FUNCTION_BLOCK Path EXTENDS Spline
VAR_INPUT
	waypointListRaw: 	ARRAY [0..100] OF RobotPoseSimple;
	radius: 			LREAL;
	thetaDZ: 				LREAL := 0.1;
END_VAR
VAR
	waypointList: 		ARRAY [0..100] 	OF 	RobotPoseSimple;		
	subsplines: 		ARRAY [0..99] 	OF  POINTER TO Spline;
	transitions: 		ARRAY [0..99] 	OF LREAL;
	nmbOfSubsplines, nmbOfPreprocessedWaypoints:	INT;
END_VAR

preprocessWaypointlist();

nmbOfSubsplines := 2*nmbOfPreprocessedWaypoints-3;

generateSubsplines();
lengthVar := calculateLength();
calculateTransitions();

startPoint := subsplines[0]^.startPointVal;
endPoint   := subsplines[nmbOfSubsplines-1]^.endPointVal;

startPoint.theta := waypointList[0].theta;
endPoint.theta	 := waypointList[nmbOfPreprocessedWaypoints-1].theta;

(* 
Implementation of abstract Spline method.
For internal inital length calculation, should be called in the constructor => protected
*)
METHOD PROTECTED  calculateLength : LREAL
VAR_INPUT
END_VAR
VAR
	i: INT;
END_VAR
calculateLength := 0;
FOR i := 0 TO nmbOfSubsplines-1 DO
	calculateLength := calculateLength + subsplines[i]^.length;
END_FOR
END_METHOD

METHOD PRIVATE calculateTransitions
VAR_INPUT
END_VAR
VAR
	i : INT;
END_VAR
transitions[0] := 0;
FOR i := 0 TO nmbOfSubsplines-2 DO
	transitions[i+1] := transitions[i] + subsplines[i]^.length;
END_FOR
END_METHOD

(* 
Implementation of abstract Spline method.
Calculates the derivate of the spline at an arbitrary arcLength. Should be implmented for order one and two. Invalid 
orders should write a -1 in every component of the return value.
*)
METHOD  PUBLIC diff : RobotPoseSimple
VAR_INPUT
	arcLength: LREAL; //arcLength at which the corresponding derivative should be calculated
	order: INT := 1;  //optional: order of the derivate, should be implemented for 1 and 2, default: 1
END_VAR
VAR
	subspline: 				POINTER TO Spline;
	arcOffset, deltaTheta: 	LREAL;
	dPos: RobotPoseSimple;
END_VAR
getSubsplineToPoint(arcLength := arcLength,
					subspline => subspline,
					arcOffset => arcOffset);
deltaTheta:= endPoint.theta - startPoint.theta; 		
diff 		:= subspline^.diff(arcLength := arcOffset, order:= order);	
diff.theta 	:= dTheta(arcLength := arcLength, order := order);
END_METHOD

METHOD PRIVATE dTheta : LREAL
VAR_INPUT
	arcLength: LREAL;
	order: INT;
END_VAR
VAR
	deltaTheta: LREAL;
END_VAR
deltaTheta := endPoint.theta - startPoint.theta;
IF arcLength < thetaDZ  OR arcLength > lengthVar - thetaDZ THEN
	dTheta := 0;
ELSIF order = 1 THEN
	dTheta := deltaTheta/2*(pi/(lengthVar-2*thetaDZ))*SIN(pi/(lengthVar-2*thetaDZ)*(arcLength-thetaDZ));
ELSIF order = 2 THEN
	dTheta := deltaTheta/2*EXPT(pi/(lengthVar-2*thetaDZ),2)*COS(pi/(lengthVar-2*thetaDZ)*(arcLength-thetaDZ));
END_IF
END_METHOD

METHOD generateSubsplines : BOOL
VAR_INPUT
END_VAR
VAR
	linearSplines:		ARRAY [0..50] OF LinearSpline;
	bezierCurves:		ARRAY [0..49] OF BezierCurve;
		
	//xTmpLinear,yTmpLinear:    		ARRAY [0..1] OF LREAL;
	wplTmpLinear:					ARRAY [0..1] OF RobotPoseSimple;
	linearSpline: LinearSpline;
	
	//xTmpBezier,yTmpBezier:    		ARRAY [0..2] OF LREAL;
	wplTmpBezier:					ARRAY [0..2] OF RobotPoseSimple;
	bezierCurve: BezierCurve;
	
	i,j,k: INT := 0;
END_VAR
IF nmbOfSubsplines <> 1 THEN 
	FOR i := 1 TO nmbOfSubsplines BY 2 DO
	k := 0;
	//extract relevant points for bezier curve creation
	FOR j := (i-1)/2 TO (i-1)/2+2 BY 1 DO
		wplTmpBezier[k] := waypointList[j];
		k := k + 1;
	END_FOR  
	bezierCurves[(i-1)/2](waypoints:=wplTmpBezier, radius:=radius);
	subsplines[i]:= ADR(bezierCurves[(i-1)/2]);
	END_FOR
	
	//first Segment is always linear
	wplTmpLinear[0] := waypointList[0];
	wplTmpLinear[1] := subsplines[1]^.startPointVal;
	linearSplines[0](wayPoints := wplTmpLinear);
	subsplines[0] := ADR(linearSplines[0]);
	
	
	//last Segment is always linear
	wplTmpLinear[0] := subsplines[nmbOfSubsplines-2]^.endPointVal;
	wplTmpLinear[1] := waypointList[nmbOfPreprocessedWaypoints-1];
	linearSplines[(nmbOfSubsplines+1)/2](wayPoints := wplTmpLinear);
	subsplines[nmbOfSubsplines-1] := ADR(linearSplines[(nmbOfSubsplines+1)/2]);
	
	
	//generate the linear segments in between
	FOR i := 2 TO nmbOfSubsplines-2 BY 2 DO
	wplTmpLinear[0] := subsplines[i-1]^.endPointVal;
	wplTmpLinear[1] := subsplines[i+1]^.startPointVal;
	linearSplines[i/2](wayPoints := wplTmpLinear);
	subsplines[i] := ADR(linearSplines[i/2]);
	END_FOR
ELSE  //nmbOfSubsplines = 1  => only one linear Segment
	
	wplTmpLinear[0] := waypointList[0];
	wplTmpLinear[1] := waypointList[1];;
	linearSplines[0](wayPoints := wplTmpLinear);
	subsplines[0] := ADR(linearSplines[0]);
END_IF
END_METHOD

(*
Implementation of abstract Spline method.
Gets the configuration of the Spline at any given arcLength. 
*)
METHOD PUBLIC  getPoint : RobotPoseSimple
VAR_INPUT
	arcLength: LREAL; //arcLength at which the Splines configuration shall be calculated.
END_VAR
VAR
	subspline: POINTER TO Spline;
	arcOffset: LREAL;
	deltaTheta: LREAL;
END_VAR
getSubsplineToPoint(arcLength := arcLength,
					subspline => subspline,
					arcOffset => arcOffset);
getPoint := subspline^.getPoint(arcLength:= arcOffset);

deltaTheta 		:= endPoint.theta - startPoint.theta;
getPoint.theta	:= theta(arcLength := arcLength);
END_METHOD

METHOD PRIVATE getSubsplineToPoint : POINTER TO Spline
VAR_INPUT
	arcLength: LREAL;
END_VAR

VAR_OUTPUT
	subspline: 	POINTER TO Spline;
	arcOffset: 	LREAL;
	i: 			INT := 0;
END_VAR
arcOffset := arcLength;
IF arcLength >= length THEN
	arcOffset := arcLength - transitions[nmbOfSubsplines-1];
	subspline := subsplines[nmbOfSubsplines-1];
	RETURN;
END_IF

FOR i := 0 TO nmbOfSubsplines-1 DO
	IF arcOffset-subsplines[i]^.length < 0 THEN
		subspline := subsplines[i];
		EXIT;
	ELSE
		arcOffset := arcOffset -subsplines[i]^.length;
	END_IF
END_FOR
END_METHOD

METHOD getSwitchingPointIntervals : ARRAY [0..98] OF LREAL
VAR_INPUT
END_VAR
VAR
	i: INT := 0;
END_VAR
FILL(arr :=  getSwitchingPointIntervals, val := -1.0);
FOR i := 1 TO nmbOfSubsplines-1 BY 1 DO
	getSwitchingPointIntervals[i-1] := transitions[i];
END_FOR
END_METHOD

METHOD PRIVATE preprocessWaypointlist 
VAR_IN_OUT
END_VAR
VAR 
	i : 				INT 			:= 0;
	nextIDX: 			INT;
	phi1, phi2: 		LREAL;
END_VAR
waypointList[0].theta := waypointListRaw[0].theta;	
waypointList[0].y := waypointListRaw[0].y/1000;	
waypointList[0].x := waypointListRaw[0].x/1000;	
nextIDX := 1;

FOR i := 1 TO 99 DO
	//exit if last point is reached, last valid point is last point in preprocessed list
	IF waypointListRaw[i+1].x = -1 AND waypointListRaw[i+1].y = -1 THEN
		waypointList[nextIDX].theta := waypointListRaw[i].theta;	
		waypointList[nextIDX].y := waypointListRaw[i].y/1000;	
		waypointList[nextIDX].x := waypointListRaw[i].x/1000;	
		EXIT;
	END_IF	

	phi1 := ATAN2(waypointListRaw[i].y-waypointListRaw[i-1].y,waypointListRaw[i].x-waypointListRaw[i-1].x);
	phi2 := ATAN2(waypointListRaw[i+1].y-waypointListRaw[i].y,waypointListRaw[i+1].x-waypointListRaw[i].x);
	IF phi1 <> phi2 THEN
		waypointList[nextIDX].theta := waypointListRaw[i].theta;	
		waypointList[nextIDX].y := waypointListRaw[i].y/1000;	
		waypointList[nextIDX].x := waypointListRaw[i].x/1000;	
		nextIDX := nextIDX +1;
	END_IF
END_FOR
nmbOfPreprocessedWaypoints := nextIDX +1;
END_METHOD

METHOD PRIVATE theta : LREAL
VAR_INPUT
	arcLength: LREAL;
END_VAR
VAR
	deltaTheta: LREAL;
END_VAR
deltaTheta := endPoint.theta - startPoint.theta;
IF arcLength < thetaDZ THEN
	theta := startPoint.theta;
ELSIF arcLength > lengthVar - thetaDZ THEN
	theta := endPoint.theta;
ELSE
	theta := startPoint.theta + deltaTheta/2*(1-COS(pi/(lengthVar-2*thetaDZ)*(arcLength-thetaDZ)));
END_IF
END_METHOD

END_FUNCTION_BLOCK

(* stored: Version 1.1.0.1, ProductVersion 3.1.4024.11
   POU Path: Id {95fe6ec8-af15-4fc0-b4c5-550c7aba9b73}, SpecialFunc None
   Method calculateLength: Id {fa9150c3-1548-4fad-bc03-2a7bdbb95fff}
   Method calculateTransitions: Id {52dbb64c-0f38-4919-8d0f-8a50326cf34d}
   Method diff: Id {c435850d-099e-4883-9ebf-b0187bee6499}
   Method dTheta: Id {7d2d238e-6c7d-41bf-901f-e1aba91ddba5}
   Method generateSubsplines: Id {64c26576-c972-4416-a2f8-ea26c3f38e4d}
   Method getPoint: Id {edc81ff7-b7ad-4aac-a526-a3258fc65de9}
   Method getSubsplineToPoint: Id {d9693a58-8dc8-4612-b85b-8d181f60b2f3}
   Method getSwitchingPointIntervals: Id {cfaa726c-df69-48c1-84c4-a6f3a80b3d25}
   Method preprocessWaypointlist: Id {eb2abc10-4b35-4a8b-a276-447cab2534b7}
   Method theta: Id {3e06842d-afd1-418d-bfed-0a225c6266f7} *)
